{attribute addProperty BoxType "BK1250-0000-0000"}
{attribute addProperty Id "CouplerCtrlAT %I*UINT000"}
{attribute addProperty CRC "2618619800"}
{attribute addProperty SizeInBites "0"}
{attribute addProperty SizeInBytes "0"}
TYPE Outputs_9C14F798 :
STRUCT
	{attribute addProperty Name "CouplerCtrl"}
	CouplerCtrl AT %I* : UINT;
END_STRUCT
END_TYPE

(* stored: Version 1.2.0.0, ProductVersion 3.1.4024.9
   DUT Outputs_9C14F798: Id {b3084a53-4437-4602-b71b-c9a6b72f9827} *)
